// Mitsubishi GX Works2 project: exercicio pulse   PLC: Q03UDV

PROGRAM MAIN
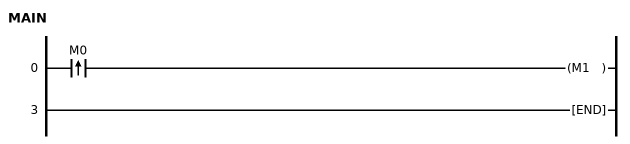
0     LDP     M0
      OUT     M1
3     END
END_PROGRAM
